FUNCTION_BLOCK BusyAgentFB (* JADE Destroyer *)
  (* Standard: 61499-1 *)
  (* Version 1.0, 2014-04-22, Ahmed, Fraunhofer IGD *)
  (* Compiler header: package fb.rt; *)
  (* Compiler Java Sun JDK 1.5.0 *)
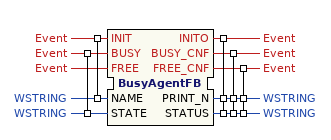
  EVENT_INPUT
    INIT WITH NAME; (* Normal Execution Request *)
    BUSY WITH STATE; (* Normal Execution Request *)
    FREE; (* Normal Execution Request *)
  END_EVENT
  EVENT_OUTPUT
    INITO WITH STATUS, PRINT_N; (* Execution Confirmation *)
    BUSY_CNF WITH PRINT_N, STATUS; (* Execution Confirmation *)
    FREE_CNF WITH STATUS, PRINT_N; (* Execution Confirmation *)
  END_EVENT
  VAR_INPUT
    NAME : WSTRING;
    STATE : WSTRING;
  END_VAR
  VAR_OUTPUT
    PRINT_N : WSTRING;
    STATUS : WSTRING;
  END_VAR
END_FUNCTION_BLOCK
